{attribute 'qualified_only'}
{attribute 'strict'}
TYPE E_MR1K1_States :
(
    Unknown := 0,
    B4C := 1,
    OUT := 2
) UINT;
END_TYPE

(* stored: Version 1.1.0.1, ProductVersion 3.1.4024.12
   DUT E_MR1K1_States: Id {b25f2d1e-112c-4694-92cb-fe3da2835bd9} *)
